{attribute 'qualified_only'}
{attribute 'strict'}
TYPE E_Color :
(
	init :=0,
	Black ,
	Red,
	Yellow,
	end
);
END_TYPE

(* stored: Version 1.1.0.1, ProductVersion 3.1.4024.12
   DUT E_Color: Id {f3e7cfd5-a5a2-43c5-bb14-5760c99b6686} *)
